# EPICS autosave request: CARSApp/Db/CARS_8_motor_settings_sub.req
# FILE... CARS_8_motor_settings_sub.req
file "CARS_motor_settings.req", P=$(P), M=$(M1)
file "CARS_motor_settings.req", P=$(P), M=$(M2)
file "CARS_motor_settings.req", P=$(P), M=$(M3)
file "CARS_motor_settings.req", P=$(P), M=$(M4)
file "CARS_motor_settings.req", P=$(P), M=$(M5)
file "CARS_motor_settings.req", P=$(P), M=$(M6)
file "CARS_motor_settings.req", P=$(P), M=$(M7)
file "CARS_motor_settings.req", P=$(P), M=$(M8)
